Omron CX-Programmer project NewProject (CX-Programmer 9.61)

# PLC NewPLC1: CP1E N30

## Global symbols (name address type ; comment)
0.00 BOOL  ; PB 1 START
100.00 BOOL  ; LAMP 1
100.01 BOOL  ; LAMP 2

## Program NewProgram1 (cyclic task 0)

### Section Section1

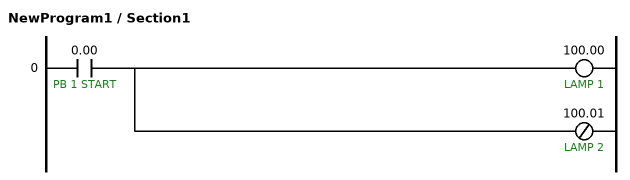
; rung 0
LD 0.00  ; PB 1 START
OUT 100.00  ; LAMP 1
OUTNOT 100.01  ; LAMP 2

### Section END
; rung 0
END(001)